{attribute 'GeneratedUsingTerminal: EL5101--0000'}
{attribute addProperty BoxType "EL5101--0000"}
{attribute addProperty Id "Channel_1AT %I*Channel_B90637B95Channel_1_1AT %Q*Channel_C6781B153WcStateAT %I*WcState_9091E0EB2InfoDataAT %I*InfoData_94A18F5E2"}
{attribute addProperty CRC "1881531089"}
{attribute addProperty Size "12"}
TYPE EL5101_7025E2D1 EXTENDS EtcSlaveTerminalBase_947E5A46 :
STRUCT
	{attribute addProperty Name "Channel_1"}
	Channel_1 : Channel_B90637B9;
	{attribute addProperty Name "Channel_1_1"}
	Channel_1_1 : Channel_C6781B15;
	{attribute addProperty Name "WcState"}
	WcState : WcState_9091E0EB;
	{attribute addProperty Name "InfoData"}
	InfoData : InfoData_94A18F5E;
END_STRUCT
END_TYPE

(* stored: Version 1.2.0.0, ProductVersion 3.1.4024.9
   DUT EL5101_7025E2D1: Id {ab7c9e3b-0523-4e0a-8584-c6a0083e480c} *)
